Fanuc KAREL source: IO_STATUS.kl

PROGRAM T
%NOLOCKGROUP
VAR
 v0 : FILE
 res : INTEGER
BEGIN
 res = IO_STATUS(v0)
END T
